Staubli VAL3: cycle_setLoop.pgx

program cycle_setLoop(bool x_bLoop (dimensions=1))
begin
  logMsg("[KERNEL] PLC:Change loop status")
  call processList:setLoop(x_bLoop)
end
